// TIA Portal project "automated_warehouse" (V18)

(* hardware
DEVICE "S7-1500/ET200MP station_1"  S7-1500 station
   slot 0: "Rail_0"  Rack  6ES7 590-1***0-0AA0
   slot 1: "PLC_1"  CPU 1511-1 PN  6ES7 511-1AL03-0AB0  V3.0
      slot 3: "CPU display_1"  6ES7591-1AA00-0AA0
      slot 32768: "PROFINET interface_1"  X1
         slot 32769: "Port_1"  X1 P1
         slot 32770: "Port_2"  X1 P2
      slot 34817: "Virtual CP interface port_1"  Virtual CP interface port  Virtual CP interface port
   slot 2: "DI 64x24VDC SNK/SRC BA_1"  DI 64x24VDC SNK/SRC BA  6ES7 521-1BP00-0AA0  V1.0
   slot 3: "DI 16x24VDC BA_1"  DI 16x24VDC BA  6ES7 521-1BH10-0AA0  V1.1
   slot 4: "DQ 64x24VDC/0.3A SNK BA_1"  DQ 64x24VDC/0.3A SNK BA  6ES7 522-1BP50-0AA0  V1.0
   slot 5: "AI 4xU/I/RTD/TC ST_1"  AI 4xU/I/RTD/TC ST  6ES7 531-7QD00-0AB0  V1.0
   slot 6: "AQ 4xU/I ST_1"  AQ 4xU/I ST  6ES7 532-5HD00-0AB0  V2.2
*)

// ===== PLC "PLC_1"  CPU 1511-1 PN =====

VAR_GLOBAL   // PLC tag table "Default tag table"
   "System_Byte" AT %MB1 : Byte;
   "FirstScan" AT %M1.0 : Bool;
   "DiagStatusUpdate" AT %M1.1 : Bool;
   "AlwaysTRUE" AT %M1.2 : Bool;
   "AlwaysFALSE" AT %M1.3 : Bool;
   "Clock_Byte" AT %MB0 : Byte;
   "Clock_10Hz" AT %M0.0 : Bool;
   "Clock_5Hz" AT %M0.1 : Bool;
   "Clock_2.5Hz" AT %M0.2 : Bool;
   "Clock_2Hz" AT %M0.3 : Bool;
   "Clock_1.25Hz" AT %M0.4 : Bool;
   "Clock_1Hz" AT %M0.5 : Bool;
   "Clock_0.625Hz" AT %M0.6 : Bool;
   "Clock_0.5Hz" AT %M0.7 : Bool;
   "Tag_1" AT %M20.0 : Bool;
END_VAR

VAR_GLOBAL   // PLC tag table "IO"
   "conv1_sensor1" AT %I0.0 : Bool;
   "conv1_sensor2" AT %I0.1 : Bool;
   "conv2_sensor1" AT %I0.2 : Bool;
   "conv2_sensor2" AT %I0.3 : Bool;
   "conv3_sensor1" AT %I0.4 : Bool;
   "conv3_sensor2" AT %I0.5 : Bool;
   "conv4_sensor1" AT %I0.6 : Bool;
   "conv4_sensor2" AT %I0.7 : Bool;
   "conv5_sensor1" AT %I1.0 : Bool;
   "conv5_sensor2" AT %I1.1 : Bool;
   "conv5_limit0" AT %I1.2 : Bool;
   "conv5_limit90" AT %I1.3 : Bool;
   "conv6_sensor1" AT %I1.4 : Bool;
   "conv6_sensor2" AT %I1.5 : Bool;
   "conv7_sensor1" AT %I1.6 : Bool;
   "conv7_sensor2" AT %I1.7 : Bool;
   "conv8_sensor1" AT %I2.0 : Bool;
   "conv8_sensor2" AT %I2.1 : Bool;
   "conv8_limit0" AT %I2.2 : Bool;
   "conv8_limit90" AT %I2.3 : Bool;
   "conv9_sensor1" AT %I2.4 : Bool;
   "conv9_sensor2" AT %I2.5 : Bool;
   "conv10_sensor1" AT %I2.6 : Bool;
   "conv10_sensor2" AT %I2.7 : Bool;
   "conv11_sensor1" AT %I3.0 : Bool;
   "conv11_sensor2" AT %I3.1 : Bool;
   "conv11_limit0" AT %I3.2 : Bool;
   "conv11_limit90" AT %I3.3 : Bool;
   "conv12_sensor1" AT %I3.4 : Bool;
   "conv12_sensor2" AT %I3.5 : Bool;
   "conv13_sensor1" AT %I3.6 : Bool;
   "conv13_sensor2" AT %I3.7 : Bool;
   "conv14_sensor1" AT %I4.0 : Bool;
   "conv14_sensor2" AT %I4.1 : Bool;
   "conv15_sensor1" AT %I4.2 : Bool;
   "conv15_sensor2" AT %I4.3 : Bool;
   "conv16_sensor1" AT %I4.4 : Bool;
   "conv16_sensor2" AT %I4.5 : Bool;
   "conv17_sensor1" AT %I4.6 : Bool;
   "conv17_sensor2" AT %I4.7 : Bool;
   "conv17_limit0" AT %I5.0 : Bool;
   "conv18_sensor1" AT %I5.2 : Bool;
   "conv18_sensor2" AT %I5.3 : Bool;
   "conv19_sensor1" AT %I5.4 : Bool;
   "conv19_sensor2" AT %I5.5 : Bool;
   "conv20_sensor1" AT %I5.6 : Bool;
   "conv20_sensor2" AT %I5.7 : Bool;
   "conv21_sensor1" AT %I6.0 : Bool;
   "conv21_sensor2" AT %I6.1 : Bool;
   "conv22_sensor1" AT %I6.2 : Bool;
   "conv22_sensor2" AT %I6.3 : Bool;
   "crane1_movingX_sensor" AT %I6.4 : Bool;
   "crane1_movingZ_sensor" AT %I6.5 : Bool;
   "fork1_load_sensor" AT %I6.6 : Bool;
   "fork1_center_sensor" AT %I6.7 : Bool;
   "fork1_unload_sensor" AT %I7.0 : Bool;
   "crane2_movingX_sensor" AT %I7.1 : Bool;
   "fork2_load_sensor" AT %I7.3 : Bool;
   "fork2_center_sensor" AT %I7.4 : Bool;
   "fork2_unload_sensor" AT %I7.5 : Bool;
   "conv1_move" AT %Q0.0 : Bool;
   "conv2_move" AT %Q0.1 : Bool;
   "conv3_move" AT %Q0.2 : Bool;
   "conv4_move" AT %Q0.3 : Bool;
   "conv5_move" AT %Q0.4 : Bool;
   "conv5_move_back" AT %Q0.5 : Bool;
   "conv5_turn" AT %Q0.6 : Bool;
   "conv6_move" AT %Q0.7 : Bool;
   "conv7_move" AT %Q1.0 : Bool;
   "conv8_move" AT %Q1.1 : Bool;
   "conv8_move_back" AT %Q1.2 : Bool;
   "conv8_turn" AT %Q1.3 : Bool;
   "conv9_move" AT %Q1.4 : Bool;
   "conv10_move" AT %Q1.5 : Bool;
   "conv11_move" AT %Q1.6 : Bool;
   "conv11_move_back" AT %Q1.7 : Bool;
   "conv11_turn" AT %Q2.0 : Bool;
   "conv12_move" AT %Q2.1 : Bool;
   "conv13_move" AT %Q2.2 : Bool;
   "conv14_move" AT %Q2.3 : Bool;
   "conv15_move" AT %Q2.4 : Bool;
   "conv16_move" AT %Q2.5 : Bool;
   "conv17_move" AT %Q2.6 : Bool;
   "conv17_move_back" AT %Q2.7 : Bool;
   "conv17_turn" AT %Q3.0 : Bool;
   "conv18_move" AT %Q3.1 : Bool;
   "conv19_move" AT %Q3.2 : Bool;
   "conv19_move_back" AT %Q3.3 : Bool;
   "conv20_move" AT %Q3.4 : Bool;
   "conv21_move" AT %Q3.5 : Bool;
   "conv22_move" AT %Q3.6 : Bool;
   "fork1_lift" AT %Q3.7 : Bool;
   "fork1_load" AT %Q4.0 : Bool;
   "fork1_unload" AT %Q4.1 : Bool;
   "fork2_lift" AT %Q4.2 : Bool;
   "fork2_load" AT %Q4.3 : Bool;
   "fork2_unload" AT %Q4.4 : Bool;
   "emitter" AT %Q4.5 : Bool;
   "remover" AT %Q4.6 : Bool;
   "RFID1_exec_command" AT %Q4.7 : Bool;
   "RFID1_read_data" AT %IW10 : Int;
   "RFID1_status" AT %IW12 : Int;
   "RFID1_command" AT %QW8 : Int;
   "conv17_limit90" AT %I5.1 : Bool;
   "conv5_height_sensor" AT %I7.6 : Bool;
   "conv5_width_sensor" AT %I7.7 : Bool;
   "RFID2_read_data" AT %IW14 : Int;
   "RFID2_status" AT %IW16 : Int;
   "conv15_height_sensor" AT %I8.0 : Bool;
   "conv15_width_sensor" AT %I8.1 : Bool;
   "conv18_height_sensor" AT %I8.2 : Bool;
   "conv18_width_sensor" AT %I8.3 : Bool;
   "RFID2_command" AT %QW10 : Int;
   "crane1_target_shelf" AT %QW12 : Int;
   "crane2_target_shelf" AT %QW14 : Int;
   "RFID2_exec_command" AT %Q5.0 : Bool;
   "crane2_movingZ_sensor" AT %I7.2 : Bool;
END_VAR

TYPE "shelf"
   STRUCT
      is_occupied : Bool;
      ID : Int;
      box_size : Int;
   END_STRUCT;
END_TYPE

TYPE "magazine_column"
   STRUCT
      shelf0 : "shelf";
      shelf1 : "shelf";
      shelf2 : "shelf";
      shelf3 : "shelf";
      shelf4 : "shelf";
      shelf5 : "shelf";
   END_STRUCT;
END_TYPE

TYPE "order"
   STRUCT
      ID : Int;
      magazine : Int;
      box_size : Int;
   END_STRUCT;
END_TYPE

DATA_BLOCK "DB"   // DB40
{ S7_Optimized_Access := 'FALSE' }
VERSION : 0.1
   VAR
      magazine1 : Array[0..8] of "magazine_column";
      magazine2 : Array[0..8] of "magazine_column";
      magazine1_Lbox_count : Int;
      magazine1_Mbox_count : Int;
      magazine1_Sbox_count : Int;
      magazine2_Lbox_count : Int;
      magazine2_Mbox_count : Int;
      magazine2_Sbox_count : Int;
      fork1_ready : Bool := true;
      fork2_ready : Bool := true;
      magazine1_quantity : Int;
      magazine2_quantity : Int;
      magazine2_conv7_quantity : Int;
      orders : Array[0..5] of "order";
      destination_magazine : Int;
      destination_target : Int;
      take_order : Bool;
   END_VAR
BEGIN
END_DATA_BLOCK

// folder: FB DBS

DATA_BLOCK "conv1_DB"   // DB1
{ S7_Optimized_Access := 'TRUE' }
VERSION : 0.1
// stored: InstanceOfName conv1
"conv1"
BEGIN
END_DATA_BLOCK

DATA_BLOCK "conv2_DB"   // DB2
{ S7_Optimized_Access := 'TRUE' }
VERSION : 0.1
// stored: InstanceOfName conv2
"conv2"
BEGIN
END_DATA_BLOCK

DATA_BLOCK "conv3_DB"   // DB3
{ S7_Optimized_Access := 'TRUE' }
VERSION : 0.1
// stored: InstanceOfName conv3
"conv3"
BEGIN
END_DATA_BLOCK

DATA_BLOCK "conv4_DB"   // DB4
{ S7_Optimized_Access := 'TRUE' }
VERSION : 0.1
// stored: InstanceOfName conv4
"conv4"
BEGIN
END_DATA_BLOCK

DATA_BLOCK "conv5_DB"   // DB5
{ S7_Optimized_Access := 'TRUE' }
VERSION : 0.1
// stored: InstanceOfName conv5
"conv5"
BEGIN
END_DATA_BLOCK

DATA_BLOCK "conv13_DB"   // DB6
{ S7_Optimized_Access := 'TRUE' }
VERSION : 0.1
// stored: InstanceOfName conv13
"conv13"
BEGIN
END_DATA_BLOCK

DATA_BLOCK "conv14_DB"   // DB7
{ S7_Optimized_Access := 'TRUE' }
VERSION : 0.1
// stored: InstanceOfName conv14
"conv14"
BEGIN
END_DATA_BLOCK

DATA_BLOCK "conv15_DB"   // DB8
{ S7_Optimized_Access := 'TRUE' }
VERSION : 0.1
// stored: InstanceOfName conv15
"conv15"
BEGIN
END_DATA_BLOCK

DATA_BLOCK "load_to_magazine_DB"   // DB9
{ S7_Optimized_Access := 'TRUE' }
VERSION : 0.1
// stored: InstanceOfName load_to_magazine
"load_to_magazine"
BEGIN
END_DATA_BLOCK

DATA_BLOCK "conv6_DB"   // DB10
{ S7_Optimized_Access := 'TRUE' }
VERSION : 0.1
// stored: InstanceOfName conv6
"conv6"
BEGIN
END_DATA_BLOCK

DATA_BLOCK "conv7_DB"   // DB11
{ S7_Optimized_Access := 'TRUE' }
VERSION : 0.1
// stored: InstanceOfName conv7
"conv7"
BEGIN
END_DATA_BLOCK

DATA_BLOCK "conv8_DB"   // DB12
{ S7_Optimized_Access := 'TRUE' }
VERSION : 0.1
// stored: InstanceOfName conv8
"conv8"
BEGIN
END_DATA_BLOCK

DATA_BLOCK "conv19_DB"   // DB13
{ S7_Optimized_Access := 'TRUE' }
VERSION : 0.1
// stored: InstanceOfName conv19
"conv19"
BEGIN
END_DATA_BLOCK

DATA_BLOCK "conv17_DB"   // DB14
{ S7_Optimized_Access := 'TRUE' }
VERSION : 0.1
// stored: InstanceOfName conv17
"conv17"
BEGIN
END_DATA_BLOCK

DATA_BLOCK "conv18_DB"   // DB15
{ S7_Optimized_Access := 'TRUE' }
VERSION : 0.1
// stored: InstanceOfName conv18
"conv18"
BEGIN
END_DATA_BLOCK

DATA_BLOCK "load_to_magazine_DB_1"   // DB16
{ S7_Optimized_Access := 'TRUE' }
VERSION : 0.1
// stored: InstanceOfName load_to_magazine
"load_to_magazine"
BEGIN
END_DATA_BLOCK

// folder: (top level)

FUNCTION_BLOCK "conv1"   // FB1, LAD
{ S7_Optimized_Access := 'TRUE' }
VERSION : 0.1
   VAR
      edge1 : Bool;
   END_VAR
   VAR_TEMP   // added for the SCL form of the ladder/FBD networks
      _w1 : Bool;
   END_VAR
BEGIN

REGION Network 1: Move forward
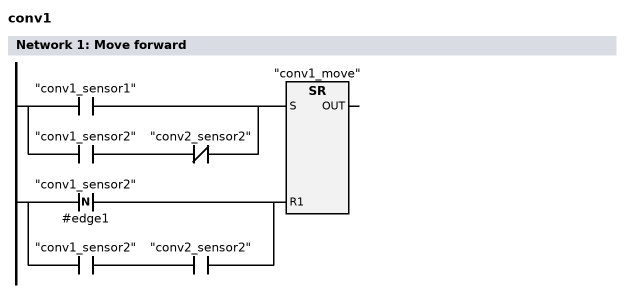
   RUNG wire#powerrail
      Contact( "conv1_sensor1" )
      wire#w1
      S_SR(operand := "conv1_move", r1 := wire#w2)
   END_RUNG
   RUNG wire#powerrail
      Contact( "conv1_sensor2" )
      I_Contact( "conv2_sensor2" )
   END_RUNG wire#w1
   RUNG wire#powerrail
      N_Contact(operand := "conv1_sensor2", bit := #edge1)
   END_RUNG wire#w2
   RUNG wire#powerrail
      Contact( "conv1_sensor2" )
      Contact( "conv2_sensor2" )
   END_RUNG wire#w2
   // the same network as SCL:
   #_w1 := NOT "conv1_sensor2" AND #edge1;   // falling edge of "conv1_sensor2"
   #edge1 := "conv1_sensor2";
   IF "conv1_sensor1" OR ("conv1_sensor2" AND NOT "conv2_sensor2") THEN
       "conv1_move" := TRUE;   // SR flip-flop
   END_IF;
   IF #_w1 OR ("conv1_sensor2" AND "conv2_sensor2") THEN "conv1_move" := FALSE; END_IF;
END_REGION
END_FUNCTION_BLOCK

FUNCTION_BLOCK "conv2"   // FB2, LAD
{ S7_Optimized_Access := 'TRUE' }
VERSION : 0.1
   VAR
      edge1 : Bool;
   END_VAR
   VAR_TEMP   // added for the SCL form of the ladder/FBD networks
      _w1 : Bool;
   END_VAR
BEGIN

REGION Network 1: Move forward
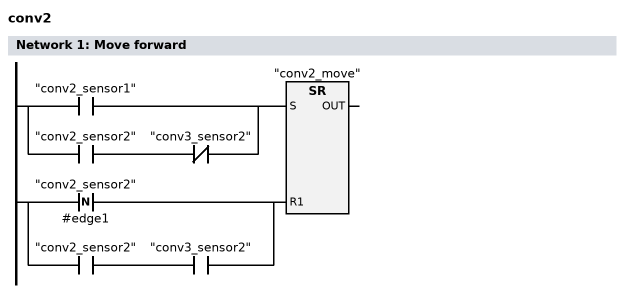
   RUNG wire#powerrail
      Contact( "conv2_sensor1" )
      wire#w1
      S_SR(operand := "conv2_move", r1 := wire#w2)
   END_RUNG
   RUNG wire#powerrail
      Contact( "conv2_sensor2" )
      I_Contact( "conv3_sensor2" )
   END_RUNG wire#w1
   RUNG wire#powerrail
      N_Contact(operand := "conv2_sensor2", bit := #edge1)
   END_RUNG wire#w2
   RUNG wire#powerrail
      Contact( "conv2_sensor2" )
      Contact( "conv3_sensor2" )
   END_RUNG wire#w2
   // the same network as SCL:
   #_w1 := NOT "conv2_sensor2" AND #edge1;   // falling edge of "conv2_sensor2"
   #edge1 := "conv2_sensor2";
   IF "conv2_sensor1" OR ("conv2_sensor2" AND NOT "conv3_sensor2") THEN
       "conv2_move" := TRUE;   // SR flip-flop
   END_IF;
   IF #_w1 OR ("conv2_sensor2" AND "conv3_sensor2") THEN "conv2_move" := FALSE; END_IF;
END_REGION
END_FUNCTION_BLOCK

FUNCTION_BLOCK "conv3"   // FB3, LAD
{ S7_Optimized_Access := 'TRUE' }
VERSION : 0.1
   VAR
      edge1 : Bool;
   END_VAR
   VAR_TEMP   // added for the SCL form of the ladder/FBD networks
      _w1 : Bool;
   END_VAR
BEGIN

REGION Network 1: Move forward
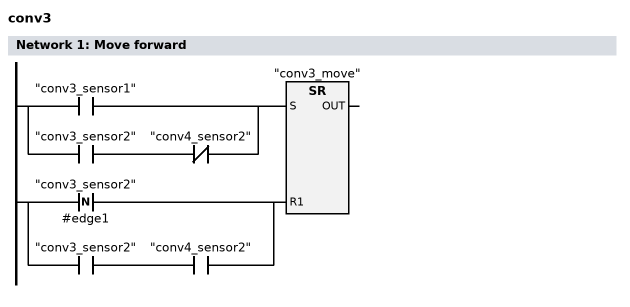
   RUNG wire#powerrail
      Contact( "conv3_sensor1" )
      wire#w1
      S_SR(operand := "conv3_move", r1 := wire#w2)
   END_RUNG
   RUNG wire#powerrail
      Contact( "conv3_sensor2" )
      I_Contact( "conv4_sensor2" )
   END_RUNG wire#w1
   RUNG wire#powerrail
      N_Contact(operand := "conv3_sensor2", bit := #edge1)
   END_RUNG wire#w2
   RUNG wire#powerrail
      Contact( "conv3_sensor2" )
      Contact( "conv4_sensor2" )
   END_RUNG wire#w2
   // the same network as SCL:
   #_w1 := NOT "conv3_sensor2" AND #edge1;   // falling edge of "conv3_sensor2"
   #edge1 := "conv3_sensor2";
   IF "conv3_sensor1" OR ("conv3_sensor2" AND NOT "conv4_sensor2") THEN
       "conv3_move" := TRUE;   // SR flip-flop
   END_IF;
   IF #_w1 OR ("conv3_sensor2" AND "conv4_sensor2") THEN "conv3_move" := FALSE; END_IF;
END_REGION
END_FUNCTION_BLOCK

FUNCTION_BLOCK "conv4"   // FB4, LAD
{ S7_Optimized_Access := 'TRUE' }
VERSION : 0.1
   VAR
      edge1 : Bool;
   END_VAR
   VAR_TEMP   // added for the SCL form of the ladder/FBD networks
      _w1 : Bool;
   END_VAR
BEGIN

REGION Network 1: Move forward
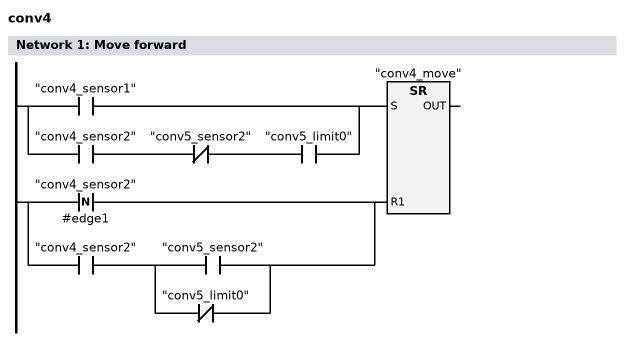
   RUNG wire#powerrail
      Contact( "conv4_sensor1" )
      wire#w1
      S_SR(operand := "conv4_move", r1 := wire#w3)
   END_RUNG
   RUNG wire#powerrail
      Contact( "conv4_sensor2" )
      I_Contact( "conv5_sensor2" )
      Contact( "conv5_limit0" )
   END_RUNG wire#w1
   RUNG wire#powerrail
      N_Contact(operand := "conv4_sensor2", bit := #edge1)
   END_RUNG wire#w3
   RUNG wire#powerrail
      Contact( "conv4_sensor2" )
      wire#w2
      Contact( "conv5_sensor2" )
   END_RUNG wire#w3
   RUNG wire#w2
      I_Contact( "conv5_limit0" )
   END_RUNG wire#w3
   // the same network as SCL:
   #_w1 := NOT "conv4_sensor2" AND #edge1;   // falling edge of "conv4_sensor2"
   #edge1 := "conv4_sensor2";
   IF "conv4_sensor1" OR ("conv4_sensor2" AND NOT "conv5_sensor2" AND "conv5_limit0") THEN
       "conv4_move" := TRUE;   // SR flip-flop
   END_IF;
   IF #_w1 OR ("conv4_sensor2" AND ("conv5_sensor2" OR NOT "conv5_limit0")) THEN
       "conv4_move" := FALSE;
   END_IF;
END_REGION
END_FUNCTION_BLOCK

FUNCTION_BLOCK "conv5"   // FB5, LAD
{ S7_Optimized_Access := 'TRUE' }
VERSION : 0.1
   VAR
      edge1 : Bool;
      edge2 : Bool;
      edge3 : Bool;
      edge4 : Bool;
      tmp1 : Bool;
      destination_magazine : Int;
      IEC_Timer_0_Instance : TON_TIME;
   END_VAR
   VAR_TEMP   // added for the SCL form of the ladder/FBD networks
      _w1 : Bool;
   END_VAR
BEGIN

REGION Network 1: Move forward
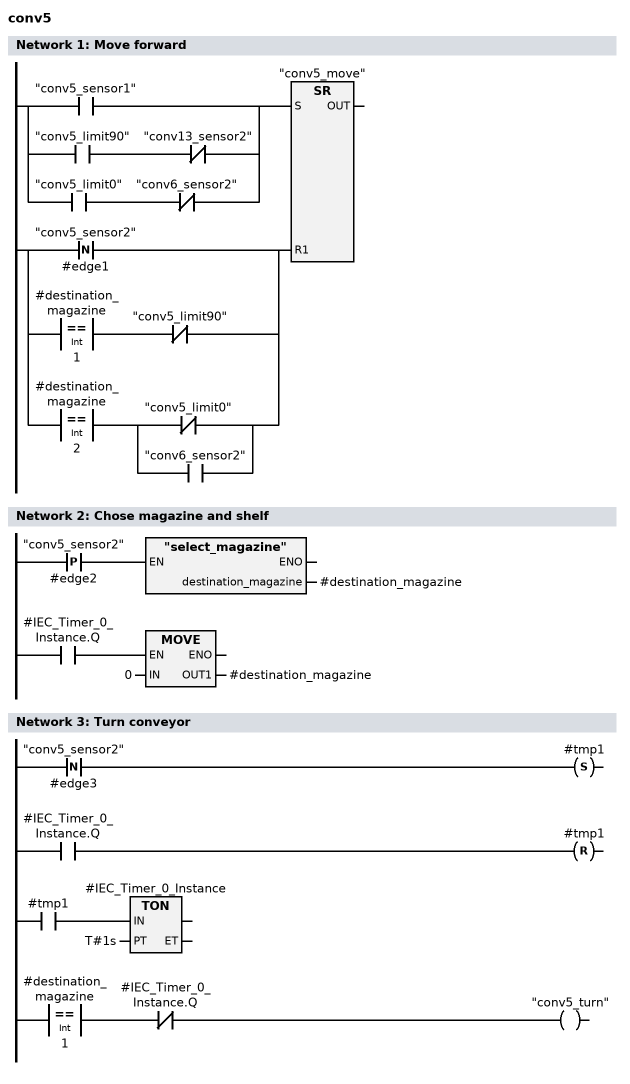
   RUNG wire#powerrail
      Contact( "conv5_sensor1" )
      wire#w1
      S_SR(operand := "conv5_move", r1 := wire#w3)
   END_RUNG
   RUNG wire#powerrail
      Contact( "conv5_limit90" )
      I_Contact( "conv13_sensor2" )
   END_RUNG wire#w1
   RUNG wire#powerrail
      Contact( "conv5_limit0" )
      I_Contact( "conv6_sensor2" )
   END_RUNG wire#w1
   RUNG wire#powerrail
      N_Contact(operand := "conv5_sensor2", bit := #edge1)
   END_RUNG wire#w3
   RUNG wire#powerrail
      { S7_Templates := "SrcType := Int" } EQ_Contact(in1 := #destination_magazine, in2 := 1)
      I_Contact( "conv5_limit90" )
   END_RUNG wire#w3
   RUNG wire#powerrail
      { S7_Templates := "SrcType := Int" } EQ_Contact(in1 := #destination_magazine, in2 := 2)
      wire#w2
      I_Contact( "conv5_limit0" )
   END_RUNG wire#w3
   RUNG wire#w2
      Contact( "conv6_sensor2" )
   END_RUNG wire#w3
   // the same network as SCL:
   #_w1 := NOT "conv5_sensor2" AND #edge1;   // falling edge of "conv5_sensor2"
   #edge1 := "conv5_sensor2";
   IF "conv5_sensor1" OR ("conv5_limit90" AND NOT "conv13_sensor2") OR ("conv5_limit0" AND NOT "conv6_sensor2") THEN
       "conv5_move" := TRUE;   // SR flip-flop
   END_IF;
   IF #_w1 OR ((#destination_magazine = 1) AND NOT "conv5_limit90") OR ((#destination_magazine = 2) AND (NOT "conv5_limit0" OR "conv6_sensor2")) THEN
       "conv5_move" := FALSE;
   END_IF;
END_REGION

REGION Network 2: Chose magazine and shelf
   RUNG wire#powerrail
      P_Contact(operand := "conv5_sensor2", bit := #edge2)
      "select_magazine"(destination_magazine => #destination_magazine)
   END_RUNG
   RUNG wire#powerrail
      Contact( #IEC_Timer_0_Instance.Q )
      Move(in := 0, out1 => #destination_magazine)
   END_RUNG
   // the same network as SCL:
   #_w1 := "conv5_sensor2" AND NOT #edge2;   // rising edge of "conv5_sensor2"
   #edge2 := "conv5_sensor2";
   IF #_w1 THEN "select_magazine"(destination_magazine => #destination_magazine); END_IF;
   IF #IEC_Timer_0_Instance.Q THEN #destination_magazine := 0; END_IF;
END_REGION

REGION Network 3: Turn conveyor
   #_w1 := NOT "conv5_sensor2" AND #edge3;   // falling edge of "conv5_sensor2"
   #edge3 := "conv5_sensor2";
   IF #_w1 THEN #tmp1 := TRUE; END_IF;
   IF #IEC_Timer_0_Instance.Q THEN #tmp1 := FALSE; END_IF;
   #IEC_Timer_0_Instance(IN := #tmp1, PT := T#1s);   // TON
   "conv5_turn" := (#destination_magazine = 1) AND NOT #IEC_Timer_0_Instance.Q;
END_REGION
END_FUNCTION_BLOCK

FUNCTION_BLOCK "conv6"   // FB6, LAD
{ S7_Optimized_Access := 'TRUE' }
VERSION : 0.1
   VAR
      edge1 : Bool;
   END_VAR
   VAR_TEMP   // added for the SCL form of the ladder/FBD networks
      _w1 : Bool;
   END_VAR
BEGIN

REGION Network 1: Move forward
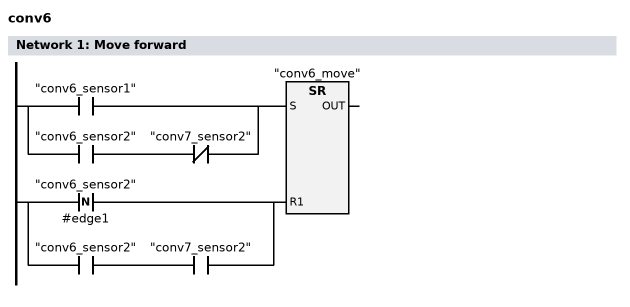
   RUNG wire#powerrail
      Contact( "conv6_sensor1" )
      wire#w1
      S_SR(operand := "conv6_move", r1 := wire#w2)
   END_RUNG
   RUNG wire#powerrail
      Contact( "conv6_sensor2" )
      I_Contact( "conv7_sensor2" )
   END_RUNG wire#w1
   RUNG wire#powerrail
      N_Contact(operand := "conv6_sensor2", bit := #edge1)
   END_RUNG wire#w2
   RUNG wire#powerrail
      Contact( "conv6_sensor2" )
      Contact( "conv7_sensor2" )
   END_RUNG wire#w2
   // the same network as SCL:
   #_w1 := NOT "conv6_sensor2" AND #edge1;   // falling edge of "conv6_sensor2"
   #edge1 := "conv6_sensor2";
   IF "conv6_sensor1" OR ("conv6_sensor2" AND NOT "conv7_sensor2") THEN
       "conv6_move" := TRUE;   // SR flip-flop
   END_IF;
   IF #_w1 OR ("conv6_sensor2" AND "conv7_sensor2") THEN "conv6_move" := FALSE; END_IF;
END_REGION
END_FUNCTION_BLOCK

FUNCTION_BLOCK "conv7"   // FB7, LAD
{ S7_Optimized_Access := 'TRUE' }
VERSION : 0.1
   VAR
      edge1 : Bool;
      edge2 : Bool;
   END_VAR
   VAR_TEMP   // added for the SCL form of the ladder/FBD networks
      _w1 : Bool;
   END_VAR
BEGIN

REGION Network 1: Move forward
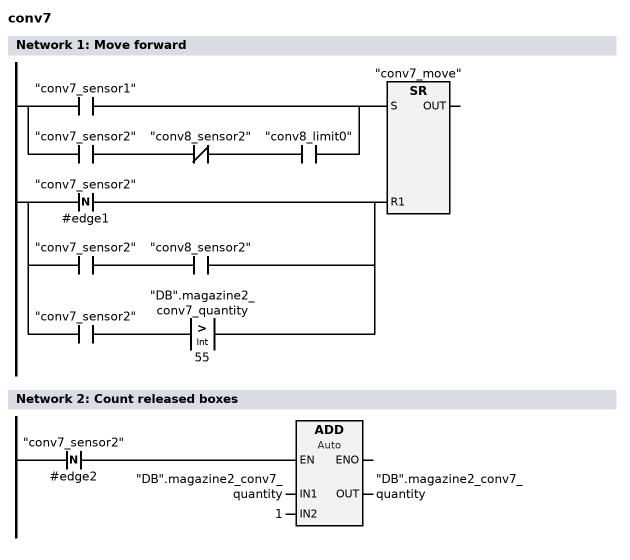
   RUNG wire#powerrail
      Contact( "conv7_sensor1" )
      wire#w1
      S_SR(operand := "conv7_move", r1 := wire#w2)
   END_RUNG
   RUNG wire#powerrail
      Contact( "conv7_sensor2" )
      I_Contact( "conv8_sensor2" )
      Contact( "conv8_limit0" )
   END_RUNG wire#w1
   RUNG wire#powerrail
      N_Contact(operand := "conv7_sensor2", bit := #edge1)
   END_RUNG wire#w2
   RUNG wire#powerrail
      Contact( "conv7_sensor2" )
      Contact( "conv8_sensor2" )
   END_RUNG wire#w2
   RUNG wire#powerrail
      Contact( "conv7_sensor2" )
      { S7_Templates := "SrcType := Int" } GT_Contact(in1 := "DB".magazine2_conv7_quantity, in2 := 55)
   END_RUNG wire#w2
   // the same network as SCL:
   #_w1 := NOT "conv7_sensor2" AND #edge1;   // falling edge of "conv7_sensor2"
   #edge1 := "conv7_sensor2";
   IF "conv7_sensor1" OR ("conv7_sensor2" AND NOT "conv8_sensor2" AND "conv8_limit0") THEN
       "conv7_move" := TRUE;   // SR flip-flop
   END_IF;
   IF #_w1 OR ("conv7_sensor2" AND "conv8_sensor2") OR ("conv7_sensor2" AND ("DB".magazine2_conv7_quantity > 55)) THEN
       "conv7_move" := FALSE;
   END_IF;
END_REGION

REGION Network 2: Count released boxes
   RUNG wire#powerrail
      N_Contact(operand := "conv7_sensor2", bit := #edge2)
      Add(in1 := "DB".magazine2_conv7_quantity, in2 := 1, out => "DB".magazine2_conv7_quantity)
   END_RUNG
   // the same network as SCL:
   #_w1 := NOT "conv7_sensor2" AND #edge2;   // falling edge of "conv7_sensor2"
   #edge2 := "conv7_sensor2";
   IF #_w1 THEN "DB".magazine2_conv7_quantity := "DB".magazine2_conv7_quantity + 1; END_IF;
END_REGION
END_FUNCTION_BLOCK

FUNCTION_BLOCK "conv8"   // FB8, LAD
{ S7_Optimized_Access := 'TRUE' }
VERSION : 0.1
   VAR
      edge1 : Bool;
      edge2 : Bool;
      tmp1 : Bool;
      IEC_Timer_0_Instance : TON_TIME;
   END_VAR
   VAR_TEMP   // added for the SCL form of the ladder/FBD networks
      _w1 : Bool;
   END_VAR
BEGIN

REGION Network 1: Move forward
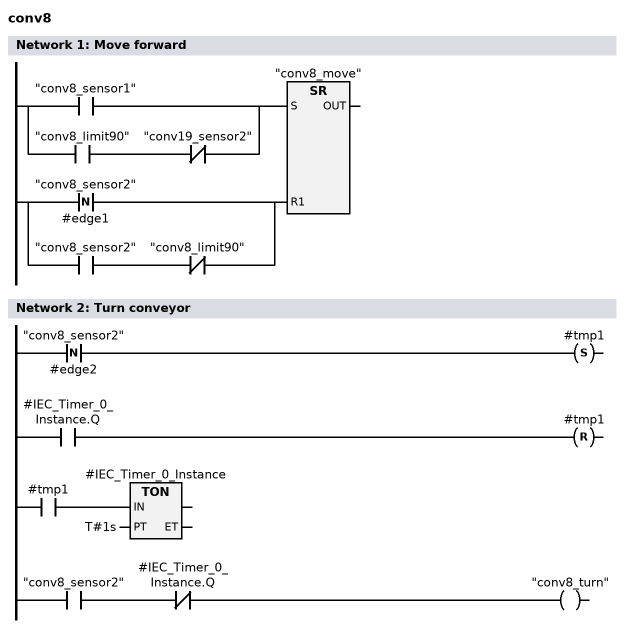
   RUNG wire#powerrail
      Contact( "conv8_sensor1" )
      wire#w1
      S_SR(operand := "conv8_move", r1 := wire#w2)
   END_RUNG
   RUNG wire#powerrail
      Contact( "conv8_limit90" )
      I_Contact( "conv19_sensor2" )
   END_RUNG wire#w1
   RUNG wire#powerrail
      N_Contact(operand := "conv8_sensor2", bit := #edge1)
   END_RUNG wire#w2
   RUNG wire#powerrail
      Contact( "conv8_sensor2" )
      I_Contact( "conv8_limit90" )
   END_RUNG wire#w2
   // the same network as SCL:
   #_w1 := NOT "conv8_sensor2" AND #edge1;   // falling edge of "conv8_sensor2"
   #edge1 := "conv8_sensor2";
   IF "conv8_sensor1" OR ("conv8_limit90" AND NOT "conv19_sensor2") THEN
       "conv8_move" := TRUE;   // SR flip-flop
   END_IF;
   IF #_w1 OR ("conv8_sensor2" AND NOT "conv8_limit90") THEN "conv8_move" := FALSE; END_IF;
END_REGION

REGION Network 2: Turn conveyor
   #_w1 := NOT "conv8_sensor2" AND #edge2;   // falling edge of "conv8_sensor2"
   #edge2 := "conv8_sensor2";
   IF #_w1 THEN #tmp1 := TRUE; END_IF;
   IF #IEC_Timer_0_Instance.Q THEN #tmp1 := FALSE; END_IF;
   #IEC_Timer_0_Instance(IN := #tmp1, PT := T#1s);   // TON
   "conv8_turn" := "conv8_sensor2" AND NOT #IEC_Timer_0_Instance.Q;
END_REGION
END_FUNCTION_BLOCK

FUNCTION_BLOCK "conv13"   // FB13, LAD
{ S7_Optimized_Access := 'TRUE' }
VERSION : 0.1
   VAR
      edge1 : Bool;
   END_VAR
   VAR_TEMP   // added for the SCL form of the ladder/FBD networks
      _w1 : Bool;
   END_VAR
BEGIN

REGION Network 1: Move forward
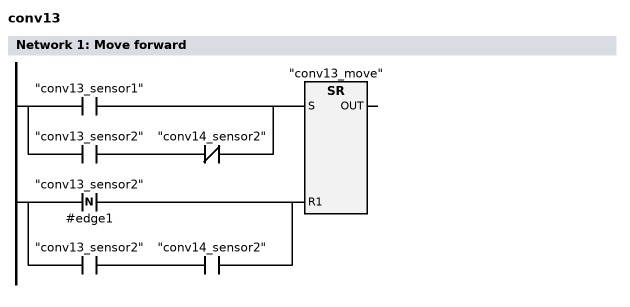
   RUNG wire#powerrail
      Contact( "conv13_sensor1" )
      wire#w1
      S_SR(operand := "conv13_move", r1 := wire#w2)
   END_RUNG
   RUNG wire#powerrail
      Contact( "conv13_sensor2" )
      I_Contact( "conv14_sensor2" )
   END_RUNG wire#w1
   RUNG wire#powerrail
      N_Contact(operand := "conv13_sensor2", bit := #edge1)
   END_RUNG wire#w2
   RUNG wire#powerrail
      Contact( "conv13_sensor2" )
      Contact( "conv14_sensor2" )
   END_RUNG wire#w2
   // the same network as SCL:
   #_w1 := NOT "conv13_sensor2" AND #edge1;   // falling edge of "conv13_sensor2"
   #edge1 := "conv13_sensor2";
   IF "conv13_sensor1" OR ("conv13_sensor2" AND NOT "conv14_sensor2") THEN
       "conv13_move" := TRUE;   // SR flip-flop
   END_IF;
   IF #_w1 OR ("conv13_sensor2" AND "conv14_sensor2") THEN "conv13_move" := FALSE; END_IF;
END_REGION
END_FUNCTION_BLOCK

FUNCTION_BLOCK "conv14"   // FB14, LAD
{ S7_Optimized_Access := 'TRUE' }
VERSION : 0.1
   VAR
      edge1 : Bool;
   END_VAR
   VAR_TEMP   // added for the SCL form of the ladder/FBD networks
      _w1 : Bool;
   END_VAR
BEGIN

REGION Network 1: Move forward
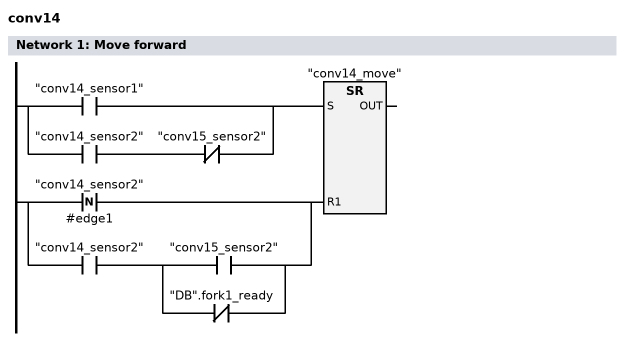
   RUNG wire#powerrail
      Contact( "conv14_sensor1" )
      wire#w1
      S_SR(operand := "conv14_move", r1 := wire#w3)
   END_RUNG
   RUNG wire#powerrail
      Contact( "conv14_sensor2" )
      I_Contact( "conv15_sensor2" )
   END_RUNG wire#w1
   RUNG wire#powerrail
      N_Contact(operand := "conv14_sensor2", bit := #edge1)
   END_RUNG wire#w3
   RUNG wire#powerrail
      Contact( "conv14_sensor2" )
      wire#w2
      Contact( "conv15_sensor2" )
   END_RUNG wire#w3
   RUNG wire#w2
      I_Contact( "DB".fork1_ready )
   END_RUNG wire#w3
   // the same network as SCL:
   #_w1 := NOT "conv14_sensor2" AND #edge1;   // falling edge of "conv14_sensor2"
   #edge1 := "conv14_sensor2";
   IF "conv14_sensor1" OR ("conv14_sensor2" AND NOT "conv15_sensor2") THEN
       "conv14_move" := TRUE;   // SR flip-flop
   END_IF;
   IF #_w1 OR ("conv14_sensor2" AND ("conv15_sensor2" OR NOT "DB".fork1_ready)) THEN
       "conv14_move" := FALSE;
   END_IF;
END_REGION
END_FUNCTION_BLOCK

FUNCTION_BLOCK "conv15"   // FB15, LAD
{ S7_Optimized_Access := 'TRUE' }
VERSION : 0.1
   VAR
      tmp1 : Bool;
      tmp2 : Bool;
      tmp3 : Bool;
      box_size : Int;
      destination_target : Int;
      step_number : Int;
      IEC_Timer_0_Instance : TON_TIME;
      IEC_Timer_0_Instance_1 : TON_TIME;
   END_VAR
   VAR_TEMP   // added for the SCL form of the ladder/FBD networks
      _w1 : Bool;
   END_VAR
BEGIN

REGION Network 1: Move forward
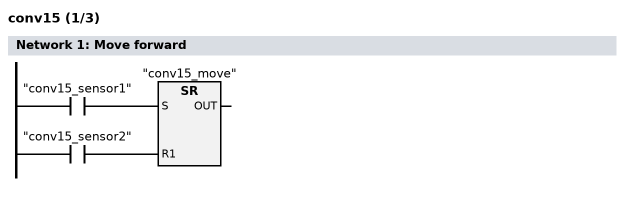
   RUNG wire#powerrail
      Contact( "conv15_sensor1" )
      S_SR(operand := "conv15_move", r1 := wire#w1)
   END_RUNG
   RUNG wire#powerrail
      Contact( "conv15_sensor2" )
   END_RUNG wire#w1
   // the same network as SCL:
   IF "conv15_sensor1" THEN
       "conv15_move" := TRUE;   // SR flip-flop
   END_IF;
   IF "conv15_sensor2" THEN "conv15_move" := FALSE; END_IF;
END_REGION

REGION Network 2: RFID read and magazine sequence
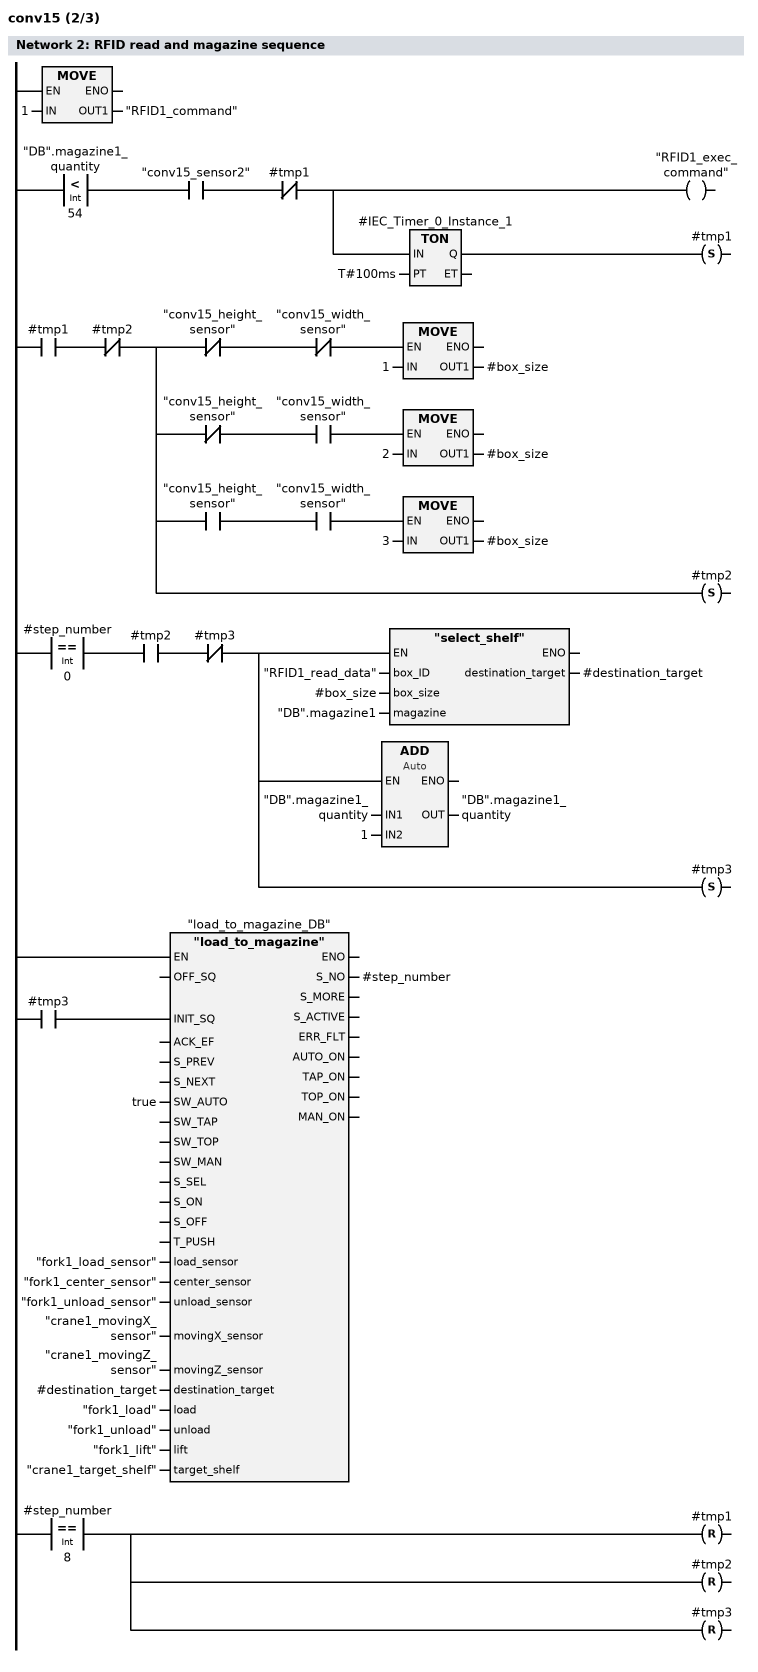
   "RFID1_command" := 1;
   "RFID1_exec_command" := ("DB".magazine1_quantity < 54) AND "conv15_sensor2" AND NOT #tmp1;
   #IEC_Timer_0_Instance_1(IN := "RFID1_exec_command", PT := T#100ms);   // TON
   IF #IEC_Timer_0_Instance_1.Q THEN #tmp1 := TRUE; END_IF;
   #_w1 := #tmp1 AND NOT #tmp2;
   IF #_w1 AND NOT "conv15_height_sensor" AND NOT "conv15_width_sensor" THEN #box_size := 1; END_IF;
   IF #_w1 AND NOT "conv15_height_sensor" AND "conv15_width_sensor" THEN #box_size := 2; END_IF;
   IF #_w1 AND "conv15_height_sensor" AND "conv15_width_sensor" THEN #box_size := 3; END_IF;
   IF #_w1 THEN #tmp2 := TRUE; END_IF;
   IF (#step_number = 0) AND #tmp2 AND NOT #tmp3 THEN
       "select_shelf"(box_ID := "RFID1_read_data",
                      box_size := #box_size,
                      magazine := "DB".magazine1,
                      destination_target => #destination_target);
       "DB".magazine1_quantity := "DB".magazine1_quantity + 1;
       #tmp3 := TRUE;
   END_IF;
   "load_to_magazine_DB"(INIT_SQ := #tmp3,   // "load_to_magazine"
                         SW_AUTO := true,
                         load_sensor := "fork1_load_sensor",
                         center_sensor := "fork1_center_sensor",
                         unload_sensor := "fork1_unload_sensor",
                         movingX_sensor := "crane1_movingX_sensor",
                         movingZ_sensor := "crane1_movingZ_sensor",
                         destination_target := #destination_target,
                         load := "fork1_load",
                         unload := "fork1_unload",
                         lift := "fork1_lift",
                         target_shelf := "crane1_target_shelf",
                         S_NO => #step_number);
   IF #step_number = 8 THEN
       #tmp1 := FALSE;
       #tmp2 := FALSE;
       #tmp3 := FALSE;
   END_IF;
END_REGION

REGION Network 3: Fork ready
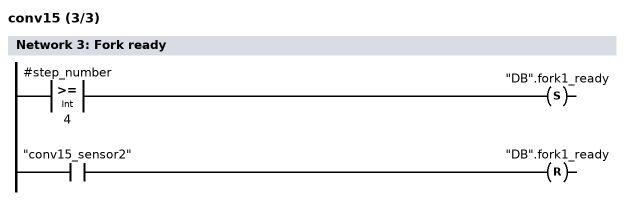
   RUNG wire#powerrail
      { S7_Templates := "SrcType := Int" } GE_Contact(in1 := #step_number, in2 := 4)
      S_Coil( "DB".fork1_ready )
   END_RUNG
   RUNG wire#powerrail
      Contact( "conv15_sensor2" )
      R_Coil( "DB".fork1_ready )
   END_RUNG
   // the same network as SCL:
   IF #step_number >= 4 THEN "DB".fork1_ready := TRUE; END_IF;
   IF "conv15_sensor2" THEN "DB".fork1_ready := FALSE; END_IF;
END_REGION
END_FUNCTION_BLOCK

FUNCTION_BLOCK "conv17"   // FB17, LAD
{ S7_Optimized_Access := 'TRUE' }
VERSION : 0.1
   VAR
      edge1 : Bool;
      edge2 : Bool;
      edge3 : Bool;
      tmp1 : Bool;
      tmp2 : Bool;
      IEC_Timer_0_Instance : TON_TIME;
   END_VAR
   VAR_TEMP   // added for the SCL form of the ladder/FBD networks
      _w1 : Bool;
   END_VAR
BEGIN

REGION Network 1: Move backward
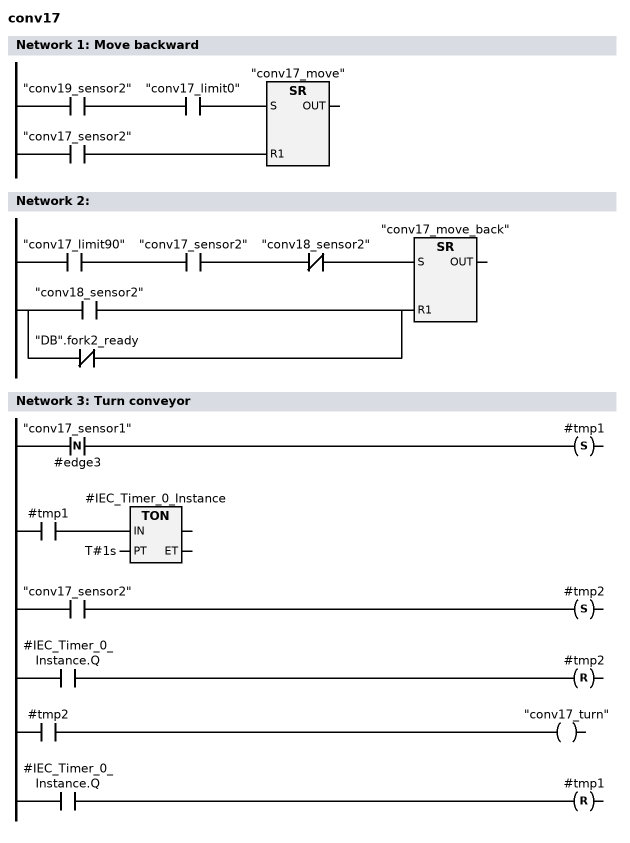
   RUNG wire#powerrail
      Contact( "conv19_sensor2" )
      Contact( "conv17_limit0" )
      S_SR(operand := "conv17_move", r1 := wire#w1)
   END_RUNG
   RUNG wire#powerrail
      Contact( "conv17_sensor2" )
   END_RUNG wire#w1
   // the same network as SCL:
   IF "conv19_sensor2" AND "conv17_limit0" THEN
       "conv17_move" := TRUE;   // SR flip-flop
   END_IF;
   IF "conv17_sensor2" THEN "conv17_move" := FALSE; END_IF;
END_REGION

REGION Network 2
   RUNG wire#powerrail
      Contact( "conv17_limit90" )
      Contact( "conv17_sensor2" )
      I_Contact( "conv18_sensor2" )
      S_SR(operand := "conv17_move_back", r1 := wire#w1)
   END_RUNG
   RUNG wire#powerrail
      Contact( "conv18_sensor2" )
   END_RUNG wire#w1
   RUNG wire#powerrail
      I_Contact( "DB".fork2_ready )
   END_RUNG wire#w1
   // the same network as SCL:
   IF "conv17_limit90" AND "conv17_sensor2" AND NOT "conv18_sensor2" THEN
       "conv17_move_back" := TRUE;   // SR flip-flop
   END_IF;
   IF "conv18_sensor2" OR NOT "DB".fork2_ready THEN "conv17_move_back" := FALSE; END_IF;
END_REGION

REGION Network 3: Turn conveyor
   #_w1 := NOT "conv17_sensor1" AND #edge3;   // falling edge of "conv17_sensor1"
   #edge3 := "conv17_sensor1";
   IF #_w1 THEN #tmp1 := TRUE; END_IF;
   #IEC_Timer_0_Instance(IN := #tmp1, PT := T#1s);   // TON
   IF "conv17_sensor2" THEN #tmp2 := TRUE; END_IF;
   IF #IEC_Timer_0_Instance.Q THEN #tmp2 := FALSE; END_IF;
   "conv17_turn" := #tmp2;
   IF #IEC_Timer_0_Instance.Q THEN #tmp1 := FALSE; END_IF;
END_REGION
END_FUNCTION_BLOCK

FUNCTION_BLOCK "conv18"   // FB18, LAD
{ S7_Optimized_Access := 'TRUE' }
VERSION : 0.1
   VAR
      tmp1 : Bool;
      tmp2 : Bool;
      tmp3 : Bool;
      box_size : Int;
      destination_target : Int;
      step_number : Int;
      IEC_Timer_0_Instance : TON_TIME;
      IEC_Timer_0_Instance_1 : TON_TIME;
   END_VAR
   VAR_TEMP   // added for the SCL form of the ladder/FBD networks
      _w1 : Bool;
   END_VAR
BEGIN

REGION Network 1: Move forward
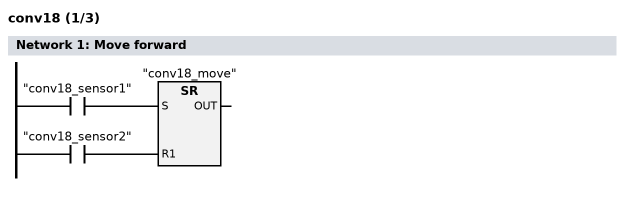
   RUNG wire#powerrail
      Contact( "conv18_sensor1" )
      S_SR(operand := "conv18_move", r1 := wire#w1)
   END_RUNG
   RUNG wire#powerrail
      Contact( "conv18_sensor2" )
   END_RUNG wire#w1
   // the same network as SCL:
   IF "conv18_sensor1" THEN
       "conv18_move" := TRUE;   // SR flip-flop
   END_IF;
   IF "conv18_sensor2" THEN "conv18_move" := FALSE; END_IF;
END_REGION

REGION Network 2: RFID read and magazine sequence
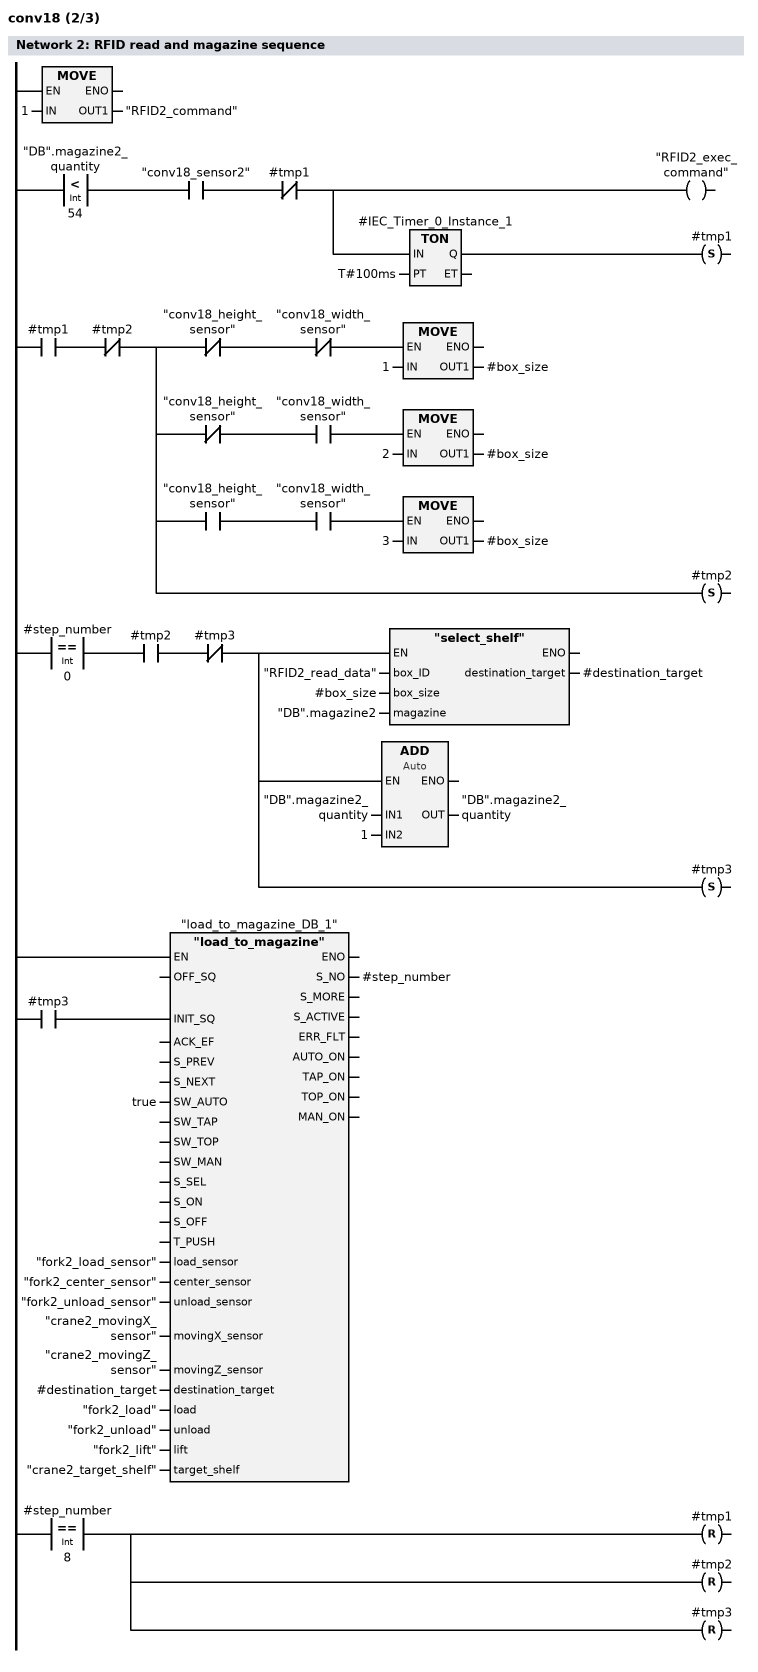
   "RFID2_command" := 1;
   "RFID2_exec_command" := ("DB".magazine2_quantity < 54) AND "conv18_sensor2" AND NOT #tmp1;
   #IEC_Timer_0_Instance_1(IN := "RFID2_exec_command", PT := T#100ms);   // TON
   IF #IEC_Timer_0_Instance_1.Q THEN #tmp1 := TRUE; END_IF;
   #_w1 := #tmp1 AND NOT #tmp2;
   IF #_w1 AND NOT "conv18_height_sensor" AND NOT "conv18_width_sensor" THEN #box_size := 1; END_IF;
   IF #_w1 AND NOT "conv18_height_sensor" AND "conv18_width_sensor" THEN #box_size := 2; END_IF;
   IF #_w1 AND "conv18_height_sensor" AND "conv18_width_sensor" THEN #box_size := 3; END_IF;
   IF #_w1 THEN #tmp2 := TRUE; END_IF;
   IF (#step_number = 0) AND #tmp2 AND NOT #tmp3 THEN
       "select_shelf"(box_ID := "RFID2_read_data",
                      box_size := #box_size,
                      magazine := "DB".magazine2,
                      destination_target => #destination_target);
       "DB".magazine2_quantity := "DB".magazine2_quantity + 1;
       #tmp3 := TRUE;
   END_IF;
   "load_to_magazine_DB_1"(INIT_SQ := #tmp3,   // "load_to_magazine"
                           SW_AUTO := true,
                           load_sensor := "fork2_load_sensor",
                           center_sensor := "fork2_center_sensor",
                           unload_sensor := "fork2_unload_sensor",
                           movingX_sensor := "crane2_movingX_sensor",
                           movingZ_sensor := "crane2_movingZ_sensor",
                           destination_target := #destination_target,
                           load := "fork2_load",
                           unload := "fork2_unload",
                           lift := "fork2_lift",
                           target_shelf := "crane2_target_shelf",
                           S_NO => #step_number);
   IF #step_number = 8 THEN
       #tmp1 := FALSE;
       #tmp2 := FALSE;
       #tmp3 := FALSE;
   END_IF;
END_REGION

REGION Network 3: Fork ready
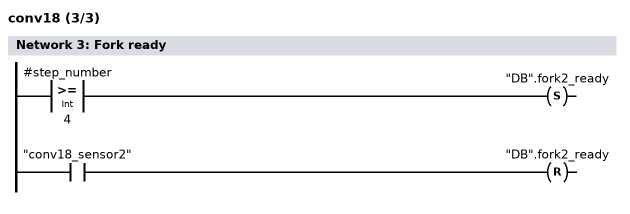
   RUNG wire#powerrail
      { S7_Templates := "SrcType := Int" } GE_Contact(in1 := #step_number, in2 := 4)
      S_Coil( "DB".fork2_ready )
   END_RUNG
   RUNG wire#powerrail
      Contact( "conv18_sensor2" )
      R_Coil( "DB".fork2_ready )
   END_RUNG
   // the same network as SCL:
   IF #step_number >= 4 THEN "DB".fork2_ready := TRUE; END_IF;
   IF "conv18_sensor2" THEN "DB".fork2_ready := FALSE; END_IF;
END_REGION
END_FUNCTION_BLOCK

FUNCTION_BLOCK "conv19"   // FB19, LAD
{ S7_Optimized_Access := 'TRUE' }
VERSION : 0.1
   VAR
      edge1 : Bool;
   END_VAR
   VAR_TEMP   // added for the SCL form of the ladder/FBD networks
      _w1 : Bool;
   END_VAR
BEGIN

REGION Network 1: Move forward
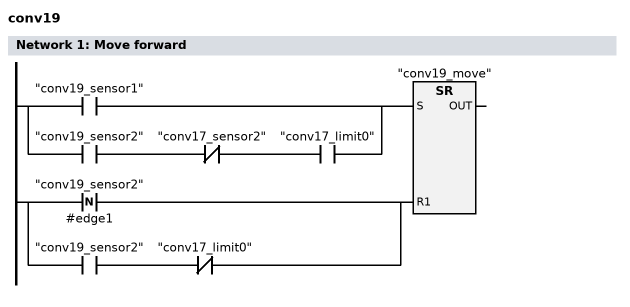
   RUNG wire#powerrail
      Contact( "conv19_sensor1" )
      wire#w1
      S_SR(operand := "conv19_move", r1 := wire#w2)
   END_RUNG
   RUNG wire#powerrail
      Contact( "conv19_sensor2" )
      I_Contact( "conv17_sensor2" )
      Contact( "conv17_limit0" )
   END_RUNG wire#w1
   RUNG wire#powerrail
      N_Contact(operand := "conv19_sensor2", bit := #edge1)
   END_RUNG wire#w2
   RUNG wire#powerrail
      Contact( "conv19_sensor2" )
      I_Contact( "conv17_limit0" )
   END_RUNG wire#w2
   // the same network as SCL:
   #_w1 := NOT "conv19_sensor2" AND #edge1;   // falling edge of "conv19_sensor2"
   #edge1 := "conv19_sensor2";
   IF "conv19_sensor1" OR ("conv19_sensor2" AND NOT "conv17_sensor2" AND "conv17_limit0") THEN
       "conv19_move" := TRUE;   // SR flip-flop
   END_IF;
   IF #_w1 OR ("conv19_sensor2" AND NOT "conv17_limit0") THEN "conv19_move" := FALSE; END_IF;
END_REGION
END_FUNCTION_BLOCK

FUNCTION_BLOCK "load_to_magazine"   // FB30, GRAPH_PLUS
{ S7_Optimized_Access := 'TRUE' }
VERSION : 0.1
   VAR_INPUT
      OFF_SQ : Bool := false;   // Turn sequence off
      INIT_SQ : Bool := false;   // Set sequence to initial state
      ACK_EF : Bool := false;   // Acknowledge all errors and faults
      S_PREV : Bool := false;   // Output previous step in parameter S_NO
      S_NEXT : Bool := false;   // Indicate next step in parameter S_NO
      SW_AUTO : Bool := false;   // Automatic mode
      SW_TAP : Bool := false;   // Semiautomatic/switch with transition
      SW_TOP : Bool := false;   // Semiautomatic/ignore transition
      SW_MAN : Bool := false;   // Manual mode
      S_SEL : Int := 0;   // Select step to be output to S_NO
      S_ON : Bool := false;   // Activate step indicated in S_NO
      S_OFF : Bool := false;   // Disable step indicated in S_NO
      T_PUSH : Bool := false;   // Enable transition to switch in semi automatic mode
      load_sensor : Bool;
      center_sensor : Bool;
      unload_sensor : Bool;
      movingX_sensor : Bool;
      movingZ_sensor : Bool;
      destination_target : Int;
   END_VAR
   VAR_OUTPUT
      S_NO : Int := 0;   // Step number
      S_MORE : Bool := false;   // More steps are available and can be shown in S_NO
      S_ACTIVE : Bool := false;   // Step indicated in S_NO is active
      ERR_FLT : Bool := false;   // Interlock or supervision group error
      AUTO_ON : Bool := false;   // Automatic mode is active
      TAP_ON : Bool := false;   // Semiautomatic mode/step with transition enabled
      TOP_ON : Bool := false;   // Semiautomatic mode/ignore transition enabled
      MAN_ON : Bool := false;   // Manual mode is active
   END_VAR
   VAR_IN_OUT
      load : Bool;
      unload : Bool;
      lift : Bool;
      target_shelf : Int;
   END_VAR
   VAR
      HMI_INFO : Array[0..8] of UInt;
      IF_PAR : G7_IfParPlus_V6;
      RT_DATA : G7_RTDataPlus_V6;   // Internal data area
      Trans1 : G7_TransitionPlus_V6;   // Transition structure
      Trans2 : G7_TransitionPlus_V6;   // Transition structure
      Trans3 : G7_TransitionPlus_V6;   // Transition structure
      Trans4 : G7_TransitionPlus_V6;   // Transition structure
      Trans5 : G7_TransitionPlus_V6;   // Transition structure
      Trans6 : G7_TransitionPlus_V6;   // Transition structure
      Trans7 : G7_TransitionPlus_V6;   // Transition structure
      Trans8 : G7_TransitionPlus_V6;   // Transition structure
      Step1 : G7_StepPlus_V6;   // Step structure
      Step2 : G7_StepPlus_V6;   // Step structure
      Step3 : G7_StepPlus_V6;   // Step structure
      Step4 : G7_StepPlus_V6;   // Step structure
      Step5 : G7_StepPlus_V6;   // Step structure
      Step6 : G7_StepPlus_V6;   // Step structure
      Step7 : G7_StepPlus_V6;   // Step structure
      Step8 : G7_StepPlus_V6;   // Step structure
      SINI : Array[0..1] of USInt;
      LSTT : Array[0..7] of USInt;
      ATAJ : Array[0..7] of USInt;
      ATAB : Array[0..7] of USInt;
      PSTT : Array[0..7] of USInt;
      NSTT : Array[0..7] of USInt;
      ASSJ : Array[0..7] of USInt;
      ASSB : Array[0..7] of USInt;
      PTTS : Array[0..7] of USInt;
      NTTS : Array[0..7] of USInt;
      SW_SQTS : Array[0..7] of USInt;
      SWITCH : Array[0..0] of USInt;
      TVX : Array[0..1] of USInt;
      TTX : Array[0..1] of USInt;
      TSX : Array[0..1] of USInt;
      S00X : Array[0..1] of USInt;
      SOFFX : Array[0..1] of USInt;
      SONX : Array[0..1] of USInt;
      SAX : Array[0..1] of USInt;
      SERRX : Array[0..8] of USInt;
      SMX : Array[0..8] of USInt;
      S0X : Array[0..8] of USInt;
      S1X : Array[0..8] of USInt;
      IL_ALARM_INST : Diag_Alarm;
      SUP_ALARM_INST : Diag_Alarm;
      STEP_TIME_ALARM_INST : Diag_Alarm;
      IEC_TIMER_INST : IEC_TIMER;
      TRANSACTION_FLAG : Bool := false;
   END_VAR
   // SINI[0] := 2;
   // LSTT[0] := 255;
   // LSTT[1] := 255;
   // LSTT[2] := 255;
   // LSTT[3] := 255;
   // LSTT[4] := 255;
   // LSTT[5] := 255;
   // LSTT[6] := 255;
   // ATAJ[1] := 1;
   // ATAJ[2] := 2;
   // ATAJ[3] := 3;
   // ATAJ[4] := 4;
   // ATAJ[5] := 5;
   // ATAJ[6] := 6;
   // ATAB[1] := 1;
   // ATAB[2] := 2;
   // ATAB[3] := 3;
   // ATAB[4] := 4;
   // ATAB[5] := 5;
   // ATAB[6] := 6;
   // PSTT[1] := 1;
   // PSTT[2] := 2;
   // PSTT[3] := 3;
   // PSTT[4] := 4;
   // PSTT[5] := 5;
   // PSTT[6] := 6;
   // NSTT[0] := 1;
   // NSTT[1] := 2;
   // NSTT[2] := 3;
   // NSTT[3] := 4;
   // NSTT[4] := 5;
   // NSTT[5] := 6;
   // NSTT[6] := 7;
   // ASSJ[1] := 1;
   // ASSJ[2] := 2;
   // ASSJ[3] := 3;
   // ASSJ[4] := 4;
   // ASSJ[5] := 5;
   // ASSJ[6] := 6;
   // ASSB[1] := 1;
   // ASSB[2] := 2;
   // ASSB[3] := 3;
   // ASSB[4] := 4;
   // ASSB[5] := 5;
   // ASSB[6] := 6;
   // PTTS[0] := 255;
   // PTTS[2] := 1;
   // PTTS[3] := 2;
   // PTTS[4] := 3;
   // PTTS[5] := 4;
   // PTTS[6] := 5;
   // NTTS[1] := 1;
   // NTTS[2] := 2;
   // NTTS[3] := 3;
   // NTTS[4] := 4;
   // NTTS[5] := 5;
   // NTTS[6] := 6;
   // TVX[0] := 16#1;
   // TTX[0] := 16#1;
   // TSX[0] := 16#1;
   // S00X[0] := 16#1;
   // SOFFX[0] := 16#1;
   // SONX[0] := 16#1;
   // SAX[0] := 16#1;
   // SERRX[0] := 16#1;
   // SMX[0] := 16#1;
   // S0X[0] := 16#1;
   // S1X[0] := 16#1;
   // LSTT[7] := 255;
   // ATAJ[7] := 7;
   // ATAB[7] := 7;
   // PSTT[7] := 7;
   // NSTT[7] := 255;
   // ASSJ[7] := 7;
   // ASSB[7] := 7;
   // PTTS[7] := 6;
   // NTTS[7] := 7;
BEGIN
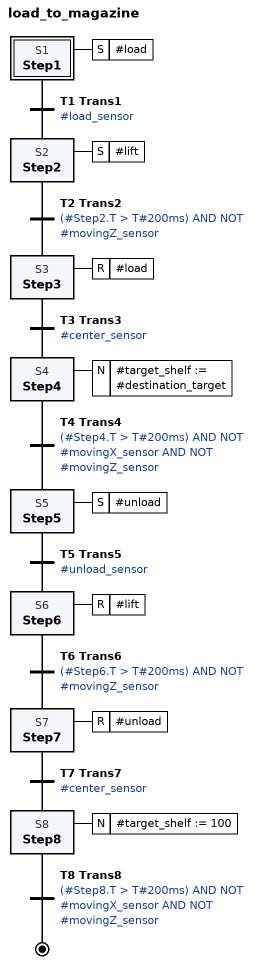
   // sequencer 1
   INITIAL_STEP Step1:   // S1, max time T#10S, warning time T#7S
              S    #load
   END_STEP
   TRANSITION Trans1 FROM Step1 TO Step2   // T1
      := #load_sensor;
   END_TRANSITION
   STEP Step2:   // S2, max time T#10S, warning time T#7S
              S    #lift
   END_STEP
   TRANSITION Trans2 FROM Step2 TO Step3   // T2
      := (#Step2.T > T#200ms) AND NOT #movingZ_sensor;
   END_TRANSITION
   STEP Step3:   // S3, max time T#10S, warning time T#7S
              R    #load
   END_STEP
   TRANSITION Trans3 FROM Step3 TO Step4   // T3
      := #center_sensor;
   END_TRANSITION
   STEP Step4:   // S4, max time T#10S, warning time T#7S
              N    #target_shelf := #destination_target
   END_STEP
   TRANSITION Trans4 FROM Step4 TO Step5   // T4
      := (#Step4.T > T#200ms) AND NOT #movingX_sensor AND NOT #movingZ_sensor;
   END_TRANSITION
   STEP Step5:   // S5, max time T#10S, warning time T#7S
              S    #unload
   END_STEP
   TRANSITION Trans5 FROM Step5 TO Step6   // T5
      := #unload_sensor;
   END_TRANSITION
   STEP Step6:   // S6, max time T#10S, warning time T#7S
              R    #lift
   END_STEP
   TRANSITION Trans6 FROM Step6 TO Step7   // T6
      := (#Step6.T > T#200ms) AND NOT #movingZ_sensor;
   END_TRANSITION
   STEP Step7:   // S7, max time T#10S, warning time T#7S
              R    #unload
   END_STEP
   TRANSITION Trans7 FROM Step7 TO Step8   // T7
      := #center_sensor;
   END_TRANSITION
   STEP Step8:   // S8, max time T#10S, warning time T#7S
              N    #target_shelf := 100
   END_STEP
   TRANSITION Trans8 FROM Step8 TO END   // T8
      := (#Step8.T > T#200ms) AND NOT #movingX_sensor AND NOT #movingZ_sensor;
   END_TRANSITION
END_FUNCTION_BLOCK

FUNCTION "select_magazine" : Void   // FC30, SCL
{ S7_Optimized_Access := 'TRUE' }
VERSION : 0.1
   VAR_OUTPUT
      destination_magazine : Int;
   END_VAR
   VAR_TEMP
      i : Int;
      box_size : Int;
   END_VAR
BEGIN
   IF "conv5_height_sensor" = FALSE AND "conv5_width_sensor" = FALSE THEN
       #box_size := 1;
   ELSIF "conv5_height_sensor" = FALSE AND "conv5_width_sensor" = TRUE THEN
       #box_size := 2;
   ELSIF "conv5_height_sensor" = TRUE AND "conv5_width_sensor" = TRUE THEN
       #box_size := 3;
   END_IF;


   IF #box_size = 1 THEN
       IF "DB".magazine1_Sbox_count <= "DB".magazine2_Sbox_count THEN
           #destination_magazine := 1;
           "DB".magazine1_Sbox_count := "DB".magazine1_Sbox_count + 1;
       ELSE
           #destination_magazine := 2;
           "DB".magazine2_Sbox_count := "DB".magazine2_Sbox_count + 1;
       END_IF;
   ELSIF #box_size = 2 THEN
       IF "DB".magazine1_Mbox_count <= "DB".magazine2_Mbox_count THEN
           #destination_magazine := 1;
           "DB".magazine1_Mbox_count := "DB".magazine1_Mbox_count + 1;
       ELSE
           #destination_magazine := 2;
           "DB".magazine2_Mbox_count := "DB".magazine2_Mbox_count + 1;
       END_IF;
   ELSIF #box_size = 3 THEN
       IF "DB".magazine1_Lbox_count <= "DB".magazine2_Lbox_count THEN
           #destination_magazine := 1;
           "DB".magazine1_Lbox_count := "DB".magazine1_Lbox_count + 1;
       ELSE
           #destination_magazine := 2;
           "DB".magazine2_Lbox_count := "DB".magazine2_Lbox_count + 1;
       END_IF;
   END_IF;
END_FUNCTION

FUNCTION "select_shelf" : Void   // FC31, SCL
{ S7_Optimized_Access := 'TRUE' }
VERSION : 0.1
   VAR_INPUT
      box_ID : Int;
      box_size : Int;
   END_VAR
   VAR_OUTPUT
      destination_target : Int;
   END_VAR
   VAR_IN_OUT
      magazine : Array[0..8] of "magazine_column";
   END_VAR
   VAR_TEMP
      i : Int;
   END_VAR
BEGIN
   FOR #i := 0 TO 8 DO
       IF #magazine[#i].shelf0.is_occupied = FALSE THEN
           #destination_target := #i + 1;

           #magazine[#i].shelf0.is_occupied := TRUE;
           #magazine[#i].shelf0.ID := #box_ID;
           #magazine[#i].shelf0.box_size := #box_size;
           EXIT;
       ELSIF #magazine[#i].shelf1.is_occupied = FALSE THEN
           #destination_target := #i + 10;

           #magazine[#i].shelf1.is_occupied := TRUE;
           #magazine[#i].shelf1.ID := #box_ID;
           #magazine[#i].shelf1.box_size := #box_size;
           EXIT;
       ELSIF #magazine[#i].shelf2.is_occupied = FALSE THEN
           #destination_target := #i + 19;

           #magazine[#i].shelf2.is_occupied := TRUE;
           #magazine[#i].shelf2.ID := #box_ID;
           #magazine[#i].shelf2.box_size := #box_size;
           EXIT;
       ELSIF #magazine[#i].shelf3.is_occupied = FALSE THEN
           #destination_target := #i + 28;

           #magazine[#i].shelf3.is_occupied := TRUE;
           #magazine[#i].shelf3.ID := #box_ID;
           #magazine[#i].shelf3.box_size := #box_size;
           EXIT;
       ELSIF #magazine[#i].shelf4.is_occupied = FALSE THEN
           #destination_target := #i + 37;

           #magazine[#i].shelf4.is_occupied := TRUE;
           #magazine[#i].shelf4.ID := #box_ID;
           #magazine[#i].shelf4.box_size := #box_size;
           EXIT;
       ELSIF #magazine[#i].shelf5.is_occupied = FALSE THEN
           #destination_target := #i + 46;

           #magazine[#i].shelf5.is_occupied := TRUE;
           #magazine[#i].shelf5.ID := #box_ID;
           #magazine[#i].shelf5.box_size := #box_size;
           EXIT;
       ELSE
           #destination_target := 100;
       END_IF;
   END_FOR;
END_FUNCTION

FUNCTION "take_order" : Void   // FC32, SCL
{ S7_Optimized_Access := 'TRUE' }
VERSION : 0.1
   VAR_OUTPUT
      destination_magazine : Int;
      destination_target : Int;
   END_VAR
   VAR_TEMP
      i : Int;
      tmp : Int;
      tmp2 : Int;
      ID : Int;
      magazine_number : Int;
      box_size : Int;
      magazine : Array[0..8] of "magazine_column";
   END_VAR
BEGIN
   #ID := "DB".orders[0].ID;
   #magazine_number := "DB".orders[0].magazine;
   #box_size := "DB".orders[0].box_size;

   FOR #i := 1 TO 5 DO
       "DB".orders[#i - 1].ID := "DB".orders[#i].ID;
       "DB".orders[#i - 1].magazine := "DB".orders[#i].magazine;
       "DB".orders[#i - 1].box_size := "DB".orders[#i].box_size;
   END_FOR;

   "DB".orders[5].ID := 0;
   "DB".orders[5].magazine := 0;
   "DB".orders[5].box_size := 0;


   IF #ID <> 0 THEN
       IF #magazine_number = 1 THEN
           #magazine := "DB".magazine1;
       ELSE
           #magazine := "DB".magazine2;
       END_IF;

       #destination_magazine := #magazine_number;
       #destination_target := 0;
       FOR #i := 0 TO 8 DO
           IF #magazine[#i].shelf0.ID = #ID THEN
               #destination_target := #i + 1;

               #magazine[#i].shelf0.is_occupied := FALSE;
               #magazine[#i].shelf0.ID := 0;
               #magazine[#i].shelf0.box_size := 0;
               EXIT;
           ELSIF #magazine[#i].shelf1.ID = #ID THEN
               #destination_target := #i + 10;

               #magazine[#i].shelf1.is_occupied := FALSE;
               #magazine[#i].shelf1.ID := 0;
               #magazine[#i].shelf1.box_size := 0;
               EXIT;
           ELSIF #magazine[#i].shelf2.ID = #ID THEN
               #destination_target := #i + 19;

               #magazine[#i].shelf2.is_occupied := FALSE;
               #magazine[#i].shelf2.ID := 0;
               #magazine[#i].shelf2.box_size := 0;
               EXIT;
           ELSIF #magazine[#i].shelf3.ID = #ID THEN
               #destination_target := #i + 28;

               #magazine[#i].shelf3.is_occupied := FALSE;
               #magazine[#i].shelf3.ID := 0;
               #magazine[#i].shelf3.box_size := 0;
               EXIT;
           ELSIF #magazine[#i].shelf4.ID = #ID THEN
               #destination_target := #i + 37;

               #magazine[#i].shelf4.is_occupied := FALSE;
               #magazine[#i].shelf4.ID := 0;
               #magazine[#i].shelf4.box_size := 0;
               EXIT;
           ELSIF #magazine[#i].shelf5.ID = #ID THEN
               #destination_target := #i + 46;

               #magazine[#i].shelf5.is_occupied := FALSE;
               #magazine[#i].shelf5.ID := 0;
               #magazine[#i].shelf5.box_size := 0;
               EXIT;
           END_IF;
       END_FOR;
   ELSE
       IF #box_size = 1 THEN
           IF "DB".magazine1_Sbox_count <= "DB".magazine2_Sbox_count THEN
               #destination_magazine := 1;
               "DB".magazine1_Sbox_count := "DB".magazine1_Sbox_count - 1;

               #tmp2 := 2;
           ELSE
               #destination_magazine := 2;
               "DB".magazine2_Sbox_count := "DB".magazine2_Sbox_count - 1;

               #tmp2 := 1;
           END_IF;
       ELSIF #box_size = 2 THEN
           IF "DB".magazine1_Mbox_count <= "DB".magazine2_Mbox_count THEN
               #destination_magazine := 1;
               "DB".magazine1_Mbox_count := "DB".magazine1_Mbox_count - 1;

               #tmp2 := 2;
           ELSE
               #destination_magazine := 2;
               "DB".magazine2_Mbox_count := "DB".magazine2_Mbox_count - 1;

               #tmp2 := 1;
           END_IF;
       ELSIF #box_size = 3 THEN
           IF "DB".magazine1_Lbox_count <= "DB".magazine2_Lbox_count THEN
               #destination_magazine := 1;
               "DB".magazine1_Lbox_count := "DB".magazine1_Lbox_count - 1;

               #tmp2 := 2;
           ELSE
               #destination_magazine := 2;
               "DB".magazine2_Lbox_count := "DB".magazine2_Lbox_count - 1;

               #tmp2 := 1;
           END_IF;
       END_IF;

       IF #tmp2 = 1 THEN
           #magazine := "DB".magazine1;
       ELSIF #tmp2 = 2 THEN
           #magazine := "DB".magazine2;
       END_IF;

       IF #tmp2 = 1 OR #tmp2 = 2 THEN
           FOR #i := 0 TO 8 DO
               IF #magazine[#i].shelf0.box_size = #box_size THEN
                   #destination_target := #i + 1;

                   #magazine[#i].shelf0.is_occupied := FALSE;
                   #magazine[#i].shelf0.ID := 0;
                   #magazine[#i].shelf0.box_size := 0;
                   EXIT;
               ELSIF #magazine[#i].shelf1.box_size = #box_size THEN
                   #destination_target := #i + 10;

                   #magazine[#i].shelf1.is_occupied := FALSE;
                   #magazine[#i].shelf1.ID := 0;
                   #magazine[#i].shelf1.box_size := 0;
                   EXIT;
               ELSIF #magazine[#i].shelf2.box_size = #box_size THEN
                   #destination_target := #i + 19;

                   #magazine[#i].shelf2.is_occupied := FALSE;
                   #magazine[#i].shelf2.ID := 0;
                   #magazine[#i].shelf2.box_size := 0;
                   EXIT;
               ELSIF #magazine[#i].shelf3.box_size = #box_size THEN
                   #destination_target := #i + 28;

                   #magazine[#i].shelf3.is_occupied := FALSE;
                   #magazine[#i].shelf3.ID := 0;
                   #magazine[#i].shelf3.box_size := 0;
                   EXIT;
               ELSIF #magazine[#i].shelf4.box_size = #box_size THEN
                   #destination_target := #i + 37;

                   #magazine[#i].shelf4.is_occupied := FALSE;
                   #magazine[#i].shelf4.ID := 0;
                   #magazine[#i].shelf4.box_size := 0;
                   EXIT;
               ELSIF #magazine[#i].shelf5.box_size = #box_size THEN
                   #destination_target := #i + 46;

                   #magazine[#i].shelf5.is_occupied := FALSE;
                   #magazine[#i].shelf5.ID := 0;
                   #magazine[#i].shelf5.box_size := 0;
                   EXIT;
               END_IF;
           END_FOR;
       ELSE
           #destination_target := 0;
       END_IF;
   END_IF;
END_FUNCTION

FUNCTION "is_order" : Void   // FC33, SCL
{ S7_Optimized_Access := 'TRUE' }
VERSION : 0.1
BEGIN
   IF "DB".orders[0].ID OR  THEN
       // Statement section IF
       ;
   END_IF;
END_FUNCTION

ORGANIZATION_BLOCK "Main"   // OB1, LAD, ProgramCycle
TITLE = "Main Program Sweep (Cycle)"
{ S7_Optimized_Access := 'TRUE' }
VERSION : 0.1
   VAR_INPUT
      Initial_Call : Bool;   // Initial call of this OB
      Remanence : Bool;   // =True, if remanent data are available
   END_VAR
   VAR_TEMP   // added for the SCL form of the ladder/FBD networks
      _w1 : Bool;
      _w2 : Bool;
      _w3 : Bool;
      _w4 : Bool;
      _w5 : Bool;
      _w6 : Bool;
      _w7 : Bool;
      _w8 : Bool;
      _w9 : Bool;
      _w10 : Bool;
      _w11 : Bool;
      _w12 : Bool;
   END_VAR
BEGIN

REGION Network 1: Enable conveyors
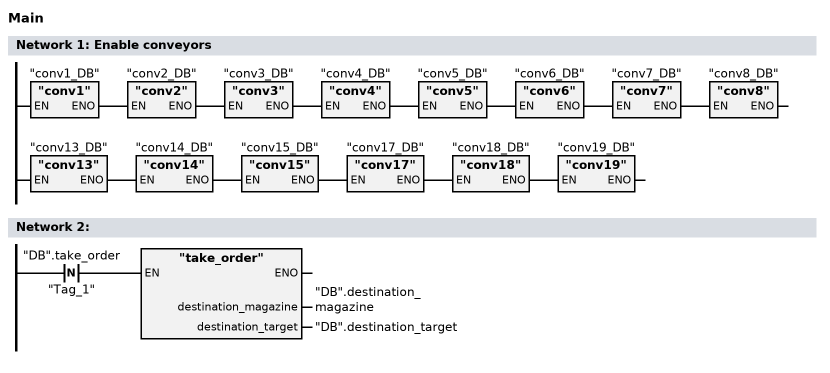
   RUNG wire#powerrail
      "conv1_DB"()
      "conv2_DB"()
      "conv3_DB"()
      "conv4_DB"()
      "conv5_DB"()
      "conv6_DB"()
      "conv7_DB"()
      "conv8_DB"()
   END_RUNG
   RUNG wire#powerrail
      "conv13_DB"()
      "conv14_DB"()
      "conv15_DB"()
      "conv17_DB"()
      "conv18_DB"()
      "conv19_DB"()
   END_RUNG
   // the same network as SCL:
   "conv1_DB"(ENO => #_w1);   // "conv1"
   "conv2_DB"(EN := #_w1, ENO => #_w2);   // "conv2"
   "conv3_DB"(EN := #_w2, ENO => #_w3);   // "conv3"
   "conv4_DB"(EN := #_w3, ENO => #_w4);   // "conv4"
   "conv5_DB"(EN := #_w4, ENO => #_w5);   // "conv5"
   "conv6_DB"(EN := #_w5, ENO => #_w6);   // "conv6"
   "conv7_DB"(EN := #_w6, ENO => #_w7);   // "conv7"
   IF #_w7 THEN
       "conv8_DB"();   // "conv8"
   END_IF;
   "conv13_DB"(ENO => #_w8);   // "conv13"
   "conv14_DB"(EN := #_w8, ENO => #_w9);   // "conv14"
   "conv15_DB"(EN := #_w9, ENO => #_w10);   // "conv15"
   "conv17_DB"(EN := #_w10, ENO => #_w11);   // "conv17"
   "conv18_DB"(EN := #_w11, ENO => #_w12);   // "conv18"
   IF #_w12 THEN
       "conv19_DB"();   // "conv19"
   END_IF;
END_REGION

REGION Network 2
   RUNG wire#powerrail
      N_Contact(operand := "DB".take_order, bit := "Tag_1")
      "take_order"(destination_magazine => "DB".destination_magazine, destination_target => "DB".destination_target)
   END_RUNG
   // the same network as SCL:
   #_w1 := NOT "DB".take_order AND "Tag_1";   // falling edge of "DB".take_order
   "Tag_1" := "DB".take_order;
   IF #_w1 THEN
       "take_order"(destination_magazine => "DB".destination_magazine,
                    destination_target => "DB".destination_target);
   END_IF;
END_REGION
END_ORGANIZATION_BLOCK